ABB RobotStudio station: Solution1_20250225-145541.rsstn

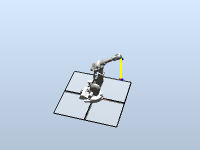
Station Solution1 (saved by RobotStudio 6.8.8148.134)
Controller R2400L
  mechanical unit ROB_1: IRB2400_10_150__02, 6 joints, base frame (0, 0, 0) mm
Layout (positions relative to the parent item):
  - IRB2400_10_150__02 [mechanism, from Robots\IRB2400_10_150_G_02.rslib] at (0, 0, 0) mm; joint values [0, 0.1639, -0.6307, 0, 1.1543, 0] (rad or m)
Targets, tools, work objects and paths stored in the station, written as RAPID:
! task T_ROB1
MODULE Module1
  CONST robtarget Target_10:=[[818.804543143,0,1822.307621556],[0.499999994,0,0.866025407,0],[0,0,0,0],[9E+09,9E+09,9E+09,9E+09,9E+09,9E+09]];
  CONST robtarget Target_20:=[[928.612158702,-400,1412.499998927],[0.499999994,0,0.866025407,0],[0,0,0,0],[9E+09,9E+09,9E+09,9E+09,9E+09,9E+09]];
  PROC Path_10()
    MoveL Target_10,v1000,z100,tool0\WObj:=wobj0;
    MoveL Target_20,v1000,z100,tool0\WObj:=wobj0;
  ENDPROC
ENDMODULE

